FUNCTION_BLOCK FB_RGBController
VAR_INPUT
END_VAR
VAR_OUTPUT
END_VAR
VAR
	iIntensityRedLED : INT;			//[0..100]
	iIntensityGreenLED : INT;
	iIntensityBlueLED : INT;
	iIntensityWhiteLED : INT;
	
	iRedLED : INT;
	iGreenLED : INT;
	iBlueLED : INT;
	iWhiteLED : INT;
END_VAR

IF iIntensityRedLED > 100 THEN
	iIntensityRedLED := iIntensityRedLED MOD 100;
END_IF
iRedLED := REAL_TO_INT(iIntensityRedLED * 0.01 * 32767);

IF iIntensityGreenLED > 100 THEN
	iIntensityGreenLED := iIntensityGreenLED MOD 100;
END_IF
iGreenLED := REAL_TO_INT(iIntensityGreenLED * 0.01 * 32767);

IF iIntensityBlueLED > 100 THEN
	iIntensityBlueLED := iIntensityBlueLED MOD 100;
END_IF
iBlueLED := REAL_TO_INT(iIntensityBlueLED * 0.01 * 32767);

IF iIntensityWhiteLED > 100 THEN
	iIntensityWhiteLED := iIntensityWhiteLED MOD 100;
END_IF
iWhiteLED := REAL_TO_INT(iIntensityWhiteLED * 0.01 * 32767);

PROPERTY setRedLED : INT
SET
END_SET
END_PROPERTY

END_FUNCTION_BLOCK

(* stored: Version 1.1.0.1, ProductVersion 3.1.4024.12
   POU FB_RGBController: Id {469ae6ce-499d-4fa3-8525-1529c7798012}, SpecialFunc None
   Property setRedLED: Id {5645f41f-39f6-4d9d-aa8e-5d7d57c0ef99}
   Set Set: Id {b79647bd-b4d7-4a42-8dd2-230e2ad1139d} *)
